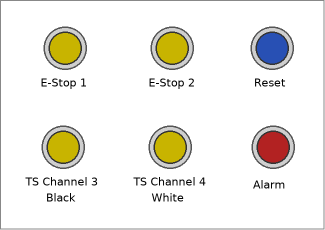
VISUALIZATION V_Safety  // 325x230
    Lamp1 (38,122 50x50), variable: TS.iSafetyMat1, style: Lamp-Lamp1-Yellow
    Lamp1 (145,122 50x50), variable: TS.iSafetyMat2, style: Lamp-Lamp1-Yellow
    Label (15,167 94x30), "TS Channel 3"
    Label (21,121 70x30)
    Label (26,183 70x30), "Black"
    Lamp1 (248,122 50x50), variable: TS.iSafetyMatAlarm, style: Lamp-Lamp1-Red
    Label (234,170 70x30), "Alarm"
    Label (123,167 94x30), "TS Channel 4"
    Label (133,183 70x30), "White"
    Lamp1 (40,23 50x50), variable: TS.iEStop1, style: Lamp-Lamp1-Yellow
    Lamp1 (147,23 50x50), variable: TS.iEStop2, style: Lamp-Lamp1-Yellow
    Label (17,68 94x30), "E-Stop 1"
    Label (125,68 94x30), "E-Stop 2"
    Lamp1 (247,23 50x50), variable: Module_IO.oResetButton, style: Lamp-Lamp1-Blue
    Label (235,68 70x30), "Reset"
END_VISUALIZATION

(* stored: Version 1.1.0.1, ProductVersion 3.1.4024.11
   Visu V_Safety: Id {61dd3f76-3f67-4346-b061-386a98d8422f} *)
